(* IEC 61131-3 sources: crb-codesys/generation/scripts/repoeval/Wrappers/PRG, 1 file *)

(* ---- PLC_PRG.st ---- *)
PROGRAM PLC_PRG
VAR
	Wrapper:FB_Wrapper;
	input: BOOL;
	output: BOOL;
END_VAR

Wrapper(in:=input , out=>output );
